Staubli VAL3: Socket1.pjx

Parameters version=s7.6 stackSize=5000 millimeterUnit=true
Program file=create.pgx
Program file=detection.pgx
Program file=getMaxNumOfPart.pgx
Program file=getObjectData.pgx
Program file=getObjectLatch.pgx
Program file=init.pgx
Program file=isDetected.pgx
Program file=kill.pgx
Program file=readSocket.pgx
Program file=readValFromSk.pgx
Program file=resetTask.pgx
Program file=start.pgx
Program file=stop.pgx
Program file=waitCharOnSk.pgx
Data file=Socket1.dtx
Library alias=ut path=Disk://Tracking/Tools/util/util.pjx
Library alias=sck path=Disk://Tracking/io/sockets/sockets.pjx
